FUNCTION_BLOCK FB_mcAxesConfigurator
VAR_INPUT
	bExecute : BOOL; // Boolean to execute the function block
	uiNoAxesRequired : UINT:= 1; // Get from user no of axes he wants to use
	sNetId: T_AmsNetId;
	pArrEcScannedSlaveInfo: POINTER TO ARRAY [0..EC_MAX_SLAVES] OF ST_EcSlaveScannedData;
	cbBufLen: UDINT;
	tTimeout: TIME;
END_VAR
VAR_OUTPUT
	uiNoAxesActive : UINT; // current no of active axes
	bNoOfAxesMatched : BOOL; // Entered no of axes matched with ECAT ring axes available
END_VAR

VAR
	uiECATScannedAxes: UINT; // Scan the ECAT ring to find the no of axis available
	fbScannedAxes	: FB_ECGETSCANNEDSLAVES;
	rTrigExecute	: R_TRIG;
END_VAR

(*Axis configurator is designed to get number of axis from user and scan ECAT 
TODO: Add further elements to it
*)

rTrigExecute(CLK:= bExecute);
M_NoOfAxes(bCommand:= rTrigExecute.Q);

METHOD M_NoOfAxes : BOOL
VAR_INPUT
	bCommand : BOOL; 
END_VAR
IF bCommand THEN

	fbScannedAxes(
		bExecute:= TRUE, 
		sNetId:= sNetId, 
		pArrEcScannedSlaveInfo:= pArrEcScannedSlaveInfo, 
		cbBufLen:= cbBufLen, 
		tTimeout:= tTimeout ,  
		nSlaves=> uiECATScannedAxes);

	IF (uiNoAxesRequired <> uiNoAxesActive) OR (uiNoAxesRequired <> uiECATScannedAxes) THEN
		
		IF (uiNoAxesRequired < mcGvl.cMinAxesCapacity) OR (uiNoAxesRequired > mcGvl.cMaxAxesCapacity) THEN
			; //TODO: Entered no of axes are not possible set the message to user
	//	ELSIF (uiNoAxesRequired <> uiECATScannedAxes) THEN
	//		bNoOfAxesMatched:=FALSE; // Entered no of axes are not matching the ECAT ring axes available
		ELSE
			uiNoAxesActive:= uiNoAxesRequired; // Set the required number of axes to active no of axes
			bNoOfAxesMatched:= TRUE;	
		END_IF
	
	ELSE
		; // cyclic calls for inequality
	END_IF
	// Reset the input of Function block so next time it has to look for only rising edge
	bExecute:= FALSE; 
ELSE
	fbScannedAxes(bExecute:= FALSE); // cyclic calls for bCommand
END_IF

M_NoOfAxes:= bNoOfAxesMatched;
END_METHOD

END_FUNCTION_BLOCK

(* stored: Version 1.1.0.1, ProductVersion 3.1.4024.6
   POU FB_mcAxesConfigurator: Id {d409f0e4-49e2-4ba1-854f-e8f860bb8e07}, SpecialFunc None
   Method M_NoOfAxes: Id {36074e18-e0b1-401a-9220-97a07c8832b3} *)
